(* CoDeSys 2.3 export: ST_TESTDATATYPE.EXP *)

(* Data type *)
(*Test comment äääöö*)
TYPE ST_TestDataType :
STRUCT
	Member : ST_Struct;
END_STRUCT
END_TYPE
